FUNCTION_BLOCK ToJSON (* Encode JSON string *)
  (* Standard: 61499-2; Description: Copyright (c) 2026 Thomas Mayr This program and the accompanying materials are made available under the terms of the Eclipse Public License 2.0 which is available at https://www.eclipse.org/legal/epl-2.0/ SPDX-License-Identifier: EPL-2.0 Adds a field to the JSONIn string. If JSONIn is empty, a new JSON object is created with the specified field. *)
  (* Version 1.0, 2026-05-16, Thomas Mayr *)
  PACKAGE eclipse4diac::convert;
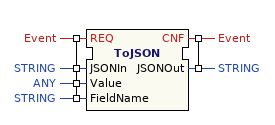
  EVENT_INPUT
    REQ WITH JSONIn, Value, FieldName; (* Execute *)
  END_EVENT
  EVENT_OUTPUT
    CNF WITH JSONOut; (* Execution done *)
  END_EVENT
  VAR_INPUT
    JSONIn : STRING; (* Input JSON string *)
    Value : ANY; (* Value to store *)
    FieldName : STRING; (* Key for the value *)
  END_VAR
  VAR_OUTPUT
    JSONOut : STRING; (* Updated JSON string *)
  END_VAR
END_FUNCTION_BLOCK
